//Main program to start MobileManipulator9DoF function block
PROGRAM MAIN
VAR
	//FB top level handler 
	fbMobileManipulator9DoF : FB_MobileManipulator9DoF;

END_VAR

fbMobileManipulator9DoF();

END_PROGRAM

(* stored: Version 1.1.0.1, ProductVersion 3.1.4024.11
   POU MAIN: Id {77c88e48-6fa6-483a-bf27-5177b3655b0b}, SpecialFunc None *)
